INTERFACE IOutputAts400 EXTENDS __SYSTEM.IQueryInterface

METHOD AbortTest
VAR_INPUT
    enable : BOOL;
END_VAR
END_METHOD

METHOD SelectProgramm : TcoCore.ITcoTaskStatus
VAR_INPUT
    programm : UINT;
END_VAR
END_METHOD

METHOD SetDummyReady
VAR_INPUT
    enable : BOOL;
END_VAR
END_METHOD

METHOD SetManualFail
VAR_INPUT
    enable : BOOL;
END_VAR
END_METHOD

METHOD SetManualPass
VAR_INPUT
    enable : BOOL;
END_VAR
END_METHOD

METHOD Start
VAR_INPUT
    enable : BOOL;
END_VAR
END_METHOD

END_INTERFACE

(* stored: Version 1.1.0.1, ProductVersion 3.1.4024.12
   Itf IOutputAts400: Id {4420b0ec-1df1-43d2-98a1-6f1a2655aaf3}
   Method AbortTest: Id {3ab7e096-3147-46cc-af48-8f13443314c0}
   Method SelectProgramm: Id {55a888aa-09eb-4122-92bb-38edb3631dfc}
   Method SetDummyReady: Id {8787423f-7186-4055-addf-3b0dfe75ceb7}
   Method SetManualFail: Id {35d1da70-7741-4c0f-bb2b-dea1c815f5f5}
   Method SetManualPass: Id {99d3b94c-f50c-404d-a69d-036e3a70f214}
   Method Start: Id {a4d5e894-7da7-4732-a9a3-d58016b687a0} *)
